FUNCTION_BLOCK AE_SPLIT_6 (* SPLIT 1 AE into 6 AE (generic FB) *)
  (* Standard: 61499-2; Description: Copyright (c) 2025 HR Agrartechnik GmbH This program and the accompanying materials are made available under the terms of the Eclipse Public License 2.0 which is available at https://www.eclipse.org/legal/epl-2.0/ SPDX-License-Identifier: EPL-2.0 *)
  (* Version 1.0, 2025-01-24, Franz Höpfinger, HR Agrartechnik GmbH *)
  PACKAGE adapter::events::unidirectional;
  IMPORT eclipse4diac::core::GenericClassName;
  IMPORT eclipse4diac::core::TypeHash;
  {SET_ATTRIBUTE(eclipse4diac::core::GenericClassName, 'GEN_AE_SPLIT')}
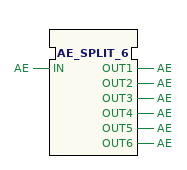
  SOCKETS
    IN : adapter::types::unidirectional::AE;
  END_SOCKETS
  PLUGS
    OUT1 : adapter::types::unidirectional::AE;
    OUT2 : adapter::types::unidirectional::AE;
    OUT3 : adapter::types::unidirectional::AE;
    OUT4 : adapter::types::unidirectional::AE;
    OUT5 : adapter::types::unidirectional::AE;
    OUT6 : adapter::types::unidirectional::AE;
  END_PLUGS
END_FUNCTION_BLOCK
